SYSTEM Test Delay
  (* Version 1.0, 2005-06-24, Goran Cengic, Chalmers *)
  DEVICE Test Device : DeviceType_not_used
    RESOURCE TestResource : ResourceType_not_used
      FBS
        restart : E_RESTART;
        merge_restart : E_MERGE2;
        merge : E_MERGE3;
        split : E_SPLIT3;
        delay3s : E_DELAY;
        delay4s : E_DELAY;
        delay5s : E_DELAY;
      END_FBS
      EVENT_CONNECTIONS
        restart.COLD TO merge_restart.EI1;
        merge_restart.EO TO split.EI;
        split.EO1 TO delay3s.START;
        split.EO2 TO delay4s.START;
        split.EO3 TO merge.EI1;
        delay3s.EO TO delay5s.STOP;
        delay4s.EO TO merge.EI3;
        merge.EO TO delay5s.START;
        delay5s.EO TO merge_restart.EI2;
      END_CONNECTIONS
      DATA_CONNECTIONS
        3000 TO delay3s.DT;
        4000 TO delay4s.DT;
        5000 TO delay5s.DT;
      END_CONNECTIONS
    END_RESOURCE
  END_DEVICE
END_SYSTEM
